PROGRAM MAIN
VAR
	
	Axis01		:		Tc2_Mc2.AXIS_REF;

END_VAR

PRG_NC_ReadWriteParameters();

END_PROGRAM

(* stored: Version 1.1.0.1, ProductVersion 3.1.4024.14
   POU MAIN: Id {f9f46e94-37ff-467b-a42a-c8c5b630cc31}, SpecialFunc None *)
